SUBAPPLICATION mapping_Uebung_049 (* DigitalInput_I1-_I4 auf DigitalOutput_Q1-_Q4 *)
  (* Standard: 61499-2; Description: Copyright (c) 2023 Meisterschulen am Ostbahnhof This program and the accompanying materials are made available under the terms of the Eclipse Public License 2.0 which is available at https://www.eclipse.org/legal/epl-2.0/ SPDX-License-Identifier: EPL-2.0 *)
  (* Version 1.0, 2023-10-23, Franz Höpfinger, Meisterschulen am Ostbahnhof *)
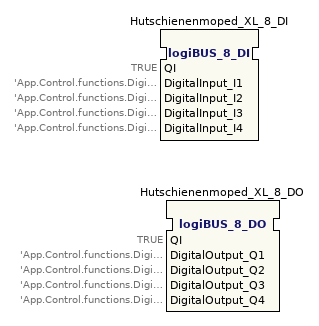
  FBS
    Hutschienenmoped_XL_8_DO : logiBUS_8_DO(QI := TRUE, DigitalOutput_Q1 := 'App.Control.functions.DigitalOutput_Q1', DigitalOutput_Q2 := 'App.Control.functions.DigitalOutput_Q2', DigitalOutput_Q3 := 'App.Control.functions.DigitalOutput_Q3', DigitalOutput_Q4 := 'App.Control.functions.DigitalOutput_Q4');
    Hutschienenmoped_XL_8_DI : logiBUS_8_DI(QI := TRUE, DigitalInput_I1 := 'App.Control.functions.DigitalInput_I1', DigitalInput_I2 := 'App.Control.functions.DigitalInput_I2', DigitalInput_I3 := 'App.Control.functions.DigitalInput_I3', DigitalInput_I4 := 'App.Control.functions.DigitalInput_I4');
  END_FBS
END_SUBAPPLICATION
